(* Logix 5000 project; controller Project1Template vendor 1 type 14 code 151 rev 33.12; software revision 33.01 *)

TASK MainTask (continuous, watchdog 500 ms) : MainProgram

MODULES
   Local : vendor 1 type 14 code 151 (Compact 0, rev 33.12)
      Discrete_IO : Embedded (Compact 1, rev 3.1, Output RPI 20 ms)
      Analog_IO : Embedded (Compact 2, rev 1.1, Output RPI 80 ms)
      Counters : Embedded (Compact 3, rev 1.1, Output RPI 20 ms)
END_MODULES

TYPE SHIFT_DATA :
STRUCT
   COMPLETED : DINT;
   PASSED : DINT;
   FAILED : DINT;
   EFFICIENT : REAL;
END_STRUCT
END_TYPE

ADD_ON_INSTRUCTION AOI_SIM_2PosCyl_ExtRet   (* revision 1.0 *)
VAR_OUTPUT
   Animation : DINT; {visible}
END_VAR
VAR_INPUT
   TravelTime : DINT; {required}
   Extend_Output : BOOL; {required}
   Retract_Output : BOOL; {required}
END_VAR
VAR_OUTPUT
   Extend_Sensor : BOOL; {access Read Only, required}
   Retract_Sensor : BOOL; {access Read Only, required}
END_VAR
VAR_INPUT
   MCR : BOOL; {required}
   SingleSolenoidExtend : BOOL; {required}
   SingleSolenoidRetract : BOOL; {required}
   Retract_ValvePB : BOOL;
   Extend_ValvePB : BOOL;
END_VAR
VAR
   Extend_ScanCount : DINT;
   Retract_ScanCount : DINT; {access None}
   Extend_Timer : TIMER := (PRE := 500); {access None}
   Retract_Timer : TIMER := (PRE := 500); {access None}
   Retracted : BOOL; {access None}
   Extended : BOOL; {access None}
   Retract : BOOL; {access None}
   Extend : BOOL; {access None}
END_VAR

ROUTINE Logic   (* ladder *)
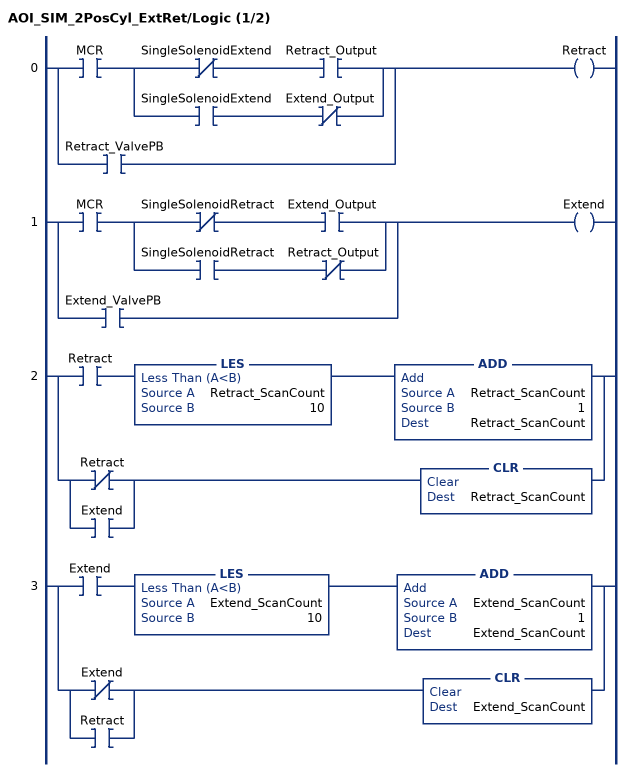
   0: [XIC(MCR) [XIO(SingleSolenoidExtend) XIC(Retract_Output) ,XIC(SingleSolenoidExtend) XIO(Extend_Output) ] ,XIC(Retract_ValvePB) ]OTE(Retract);
   1: [XIC(MCR) [XIO(SingleSolenoidRetract) XIC(Extend_Output) ,XIC(SingleSolenoidRetract) XIO(Retract_Output) ] ,XIC(Extend_ValvePB) ]OTE(Extend);
   2: [XIC(Retract) LES(Retract_ScanCount,10) ADD(Retract_ScanCount,1,Retract_ScanCount) ,[XIO(Retract) ,XIC(Extend) ] CLR(Retract_ScanCount) ];
   3: [XIC(Extend) LES(Extend_ScanCount,10) ADD(Extend_ScanCount,1,Extend_ScanCount) ,[XIO(Extend) ,XIC(Retract) ] CLR(Extend_ScanCount) ];
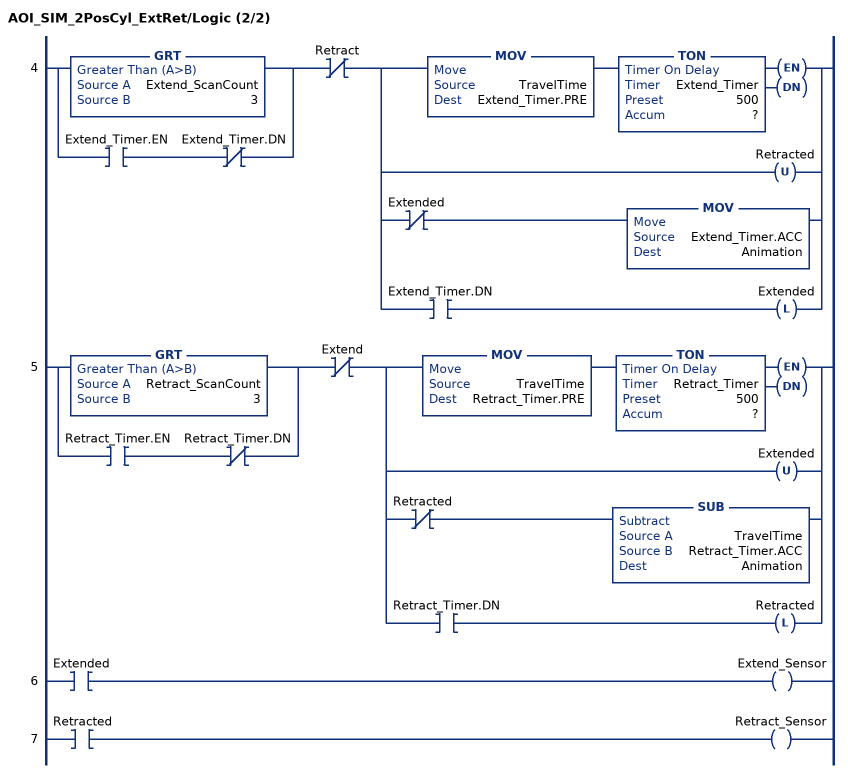
   4: [GRT(Extend_ScanCount,3) ,XIC(Extend_Timer.EN) XIO(Extend_Timer.DN) ]XIO(Retract)[MOV(TravelTime,Extend_Timer.PRE) TON(Extend_Timer,?,?) ,OTU(Retracted) ,XIO(Extended) MOV(Extend_Timer.ACC,Animation) ,XIC(Extend_Timer.DN) OTL(Extended) ];
   5: [GRT(Retract_ScanCount,3) ,XIC(Retract_Timer.EN) XIO(Retract_Timer.DN) ]XIO(Extend)[MOV(TravelTime,Retract_Timer.PRE) TON(Retract_Timer,?,?) ,OTU(Extended) ,XIO(Retracted) SUB(TravelTime,Retract_Timer.ACC,Animation) ,XIC(Retract_Timer.DN) OTL(Retracted) ];
   6: XIC(Extended)OTE(Extend_Sensor);
   7: XIC(Retracted)OTE(Retract_Sensor);
END_ROUTINE
END_ADD_ON_INSTRUCTION

ADD_ON_INSTRUCTION AOI_SIM_RandomDelay   (* revision 1.0 *)
VAR_INPUT
   Activate : BOOL; {access None}
   Target : DINT; {access None, required}
   Tolerance : DINT; {access None, required}
   PulseOutputTime : DINT; {access None, required}
END_VAR
VAR_OUTPUT
   DN : BOOL; {access Read Only, required}
END_VAR
VAR_INPUT
   DeActivate : BOOL; {access None}
END_VAR
VAR_OUTPUT
   TimingFirstHalf : BOOL; {access Read Only}
   TimingLastHalf : BOOL; {access Read Only}
   AccumlatedTime : DINT; {access Read Only}
   TT : BOOL; {access Read Only}
END_VAR
VAR
   StartTimerPulse : BOOL; {access None}
   StartTimerONS : BOOL; {access None}
   RandomIntermediate : DINT; {access None}
   RandomNumber : DINT; {access None}
   RandomPresetTime : DINT; {access None}
   RandomTimer : TIMER; {access None}
   PulseOutput : TIMER; {access None}
   Time50Percent : DINT; {access None}
END_VAR

ROUTINE Logic   (* ladder *)
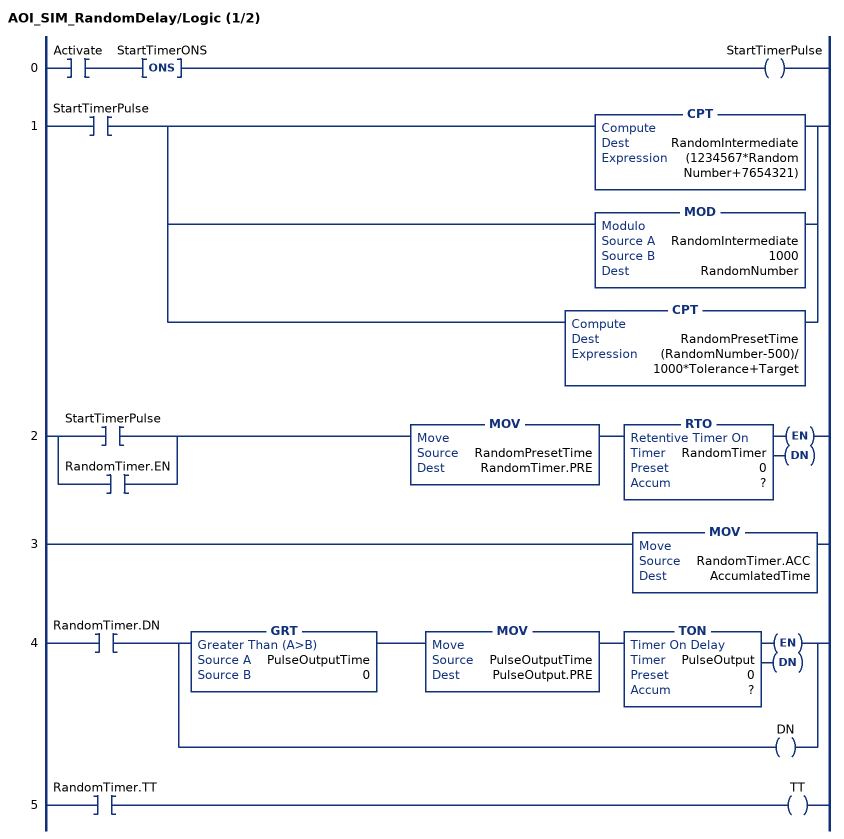
   0: XIC(Activate)ONS(StartTimerONS)OTE(StartTimerPulse);
   1: XIC(StartTimerPulse)[CPT(RandomIntermediate,(1234567*RandomNumber+7654321)) ,MOD(RandomIntermediate,1000,RandomNumber) ,CPT(RandomPresetTime,(RandomNumber-500)/1000*Tolerance+Target) ];
   2: [XIC(StartTimerPulse) ,XIC(RandomTimer.EN) ]MOV(RandomPresetTime,RandomTimer.PRE)RTO(RandomTimer,?,?);
   3: MOV(RandomTimer.ACC,AccumlatedTime);
   4: XIC(RandomTimer.DN)[GRT(PulseOutputTime,0) MOV(PulseOutputTime,PulseOutput.PRE) TON(PulseOutput,?,?) ,OTE(DN) ];
   5: XIC(RandomTimer.TT)OTE(TT);
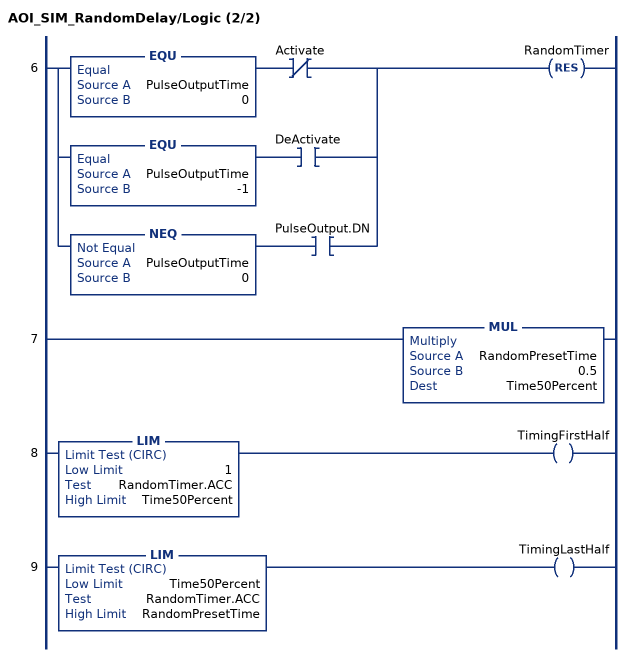
   6: [EQU(PulseOutputTime,0) XIO(Activate) ,EQU(PulseOutputTime,-1) XIC(DeActivate) ,NEQ(PulseOutputTime,0) XIC(PulseOutput.DN) ]RES(RandomTimer);
   7: MUL(RandomPresetTime,0.5,Time50Percent);
   8: LIM(1,RandomTimer.ACC,Time50Percent)OTE(TimingFirstHalf);
   9: LIM(Time50Percent,RandomTimer.ACC,RandomPresetTime)OTE(TimingLastHalf);
END_ROUTINE
END_ADD_ON_INSTRUCTION

ADD_ON_INSTRUCTION AOI_SIMAnalogSensor   (* revision 1.0 *)
VAR_IN_OUT
   Sensor : REAL; {required}
END_VAR
VAR_INPUT
   RampUpTime : DINT; {required}
   RampDwnTime : DINT; {required}
   Min : REAL; {required}
   Max : REAL; {required}
   Target : REAL; {required}
   Tolerance : REAL; {required}
   Fluctuation : REAL; {access None, required}
   Activate : BOOL; {access None}
END_VAR
VAR
   RampUpTimer : TIMER; {access None}
   RampDwnTimer : TIMER; {access None}
   FluctuateTimer : TIMER; {access None}
   FluctuateONS : BOOL; {access None}
   CurrentValue : REAL; {access Read Only}
   RampDwnTriggerONS : BOOL; {access Read Only}
   RampDwnTriggerPulse : BOOL; {access Read Only}
   RampUpTriggerONS : BOOL; {access Read Only}
   RampUpTriggerPulse : BOOL; {access Read Only}
   RandomNumber : DINT; {access Read Only}
   RandomTarget : REAL; {access Read Only}
   RandomIntermediate : DINT; {access Read Only}
   ScaledRampDwnTime : REAL; {access Read Only}
   ScaledRampUpTime : REAL; {access Read Only}
   Fluctuate : BOOL; {access None}
END_VAR

ROUTINE Logic   (* ladder *)
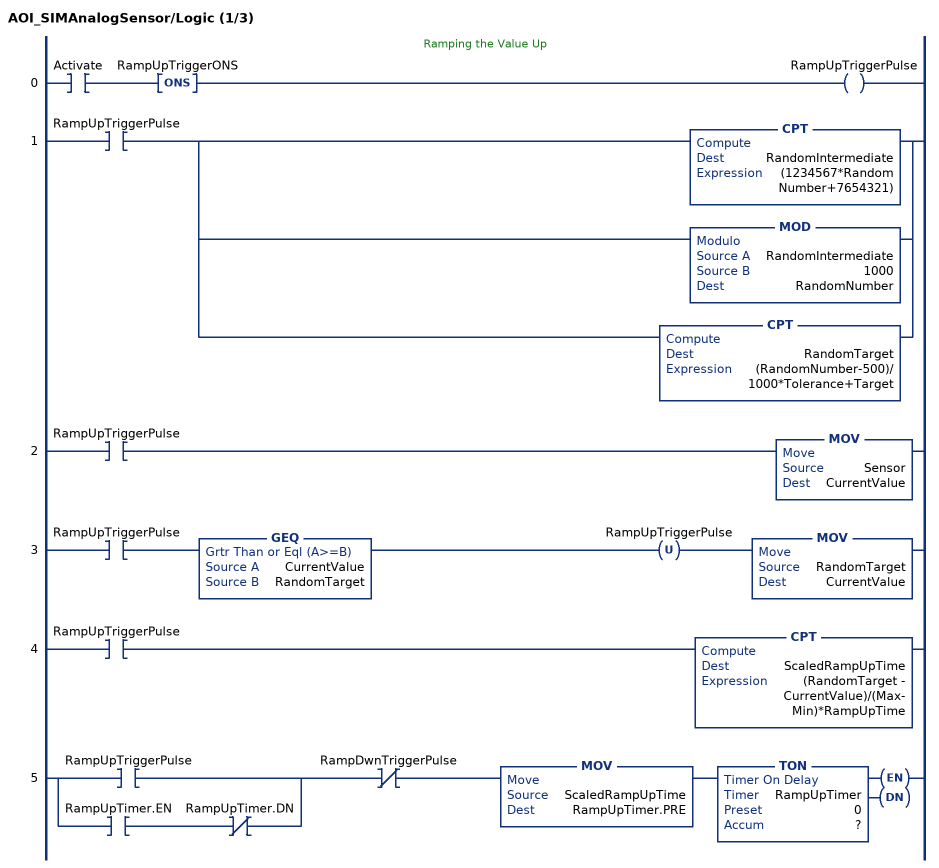
   // Ramping the Value Up
   0: XIC(Activate)ONS(RampUpTriggerONS)OTE(RampUpTriggerPulse);
   1: XIC(RampUpTriggerPulse)[CPT(RandomIntermediate,(1234567*RandomNumber+7654321)) ,MOD(RandomIntermediate,1000,RandomNumber) ,CPT(RandomTarget,(RandomNumber-500)/1000*Tolerance+Target) ];
   2: XIC(RampUpTriggerPulse)MOV(Sensor,CurrentValue);
   3: XIC(RampUpTriggerPulse)GEQ(CurrentValue,RandomTarget)OTU(RampUpTriggerPulse)MOV(RandomTarget,CurrentValue);
   4: XIC(RampUpTriggerPulse)CPT(ScaledRampUpTime,(RandomTarget - CurrentValue)/(Max-Min)*RampUpTime);
   5: [XIC(RampUpTriggerPulse) ,XIC(RampUpTimer.EN) XIO(RampUpTimer.DN) ]XIO(RampDwnTriggerPulse)MOV(ScaledRampUpTime,RampUpTimer.PRE)TON(RampUpTimer,?,?);
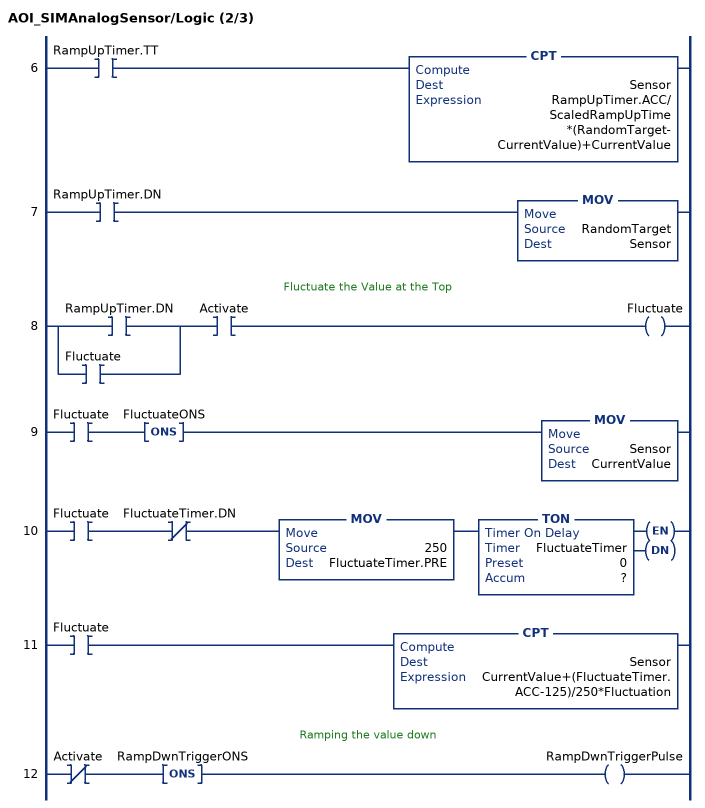
   6: XIC(RampUpTimer.TT)CPT(Sensor,RampUpTimer.ACC/ScaledRampUpTime *(RandomTarget-CurrentValue)+CurrentValue);
   7: XIC(RampUpTimer.DN)MOV(RandomTarget,Sensor);
   // Fluctuate the Value at the Top
   8: [XIC(RampUpTimer.DN) ,XIC(Fluctuate) ]XIC(Activate)OTE(Fluctuate);
   9: XIC(Fluctuate)ONS(FluctuateONS)MOV(Sensor,CurrentValue);
   10: XIC(Fluctuate)XIO(FluctuateTimer.DN)MOV(250,FluctuateTimer.PRE)TON(FluctuateTimer,?,?);
   11: XIC(Fluctuate)CPT(Sensor,CurrentValue+(FluctuateTimer.ACC-125)/250*Fluctuation);
   // Ramping the value down
   12: XIO(Activate)ONS(RampDwnTriggerONS)OTE(RampDwnTriggerPulse);
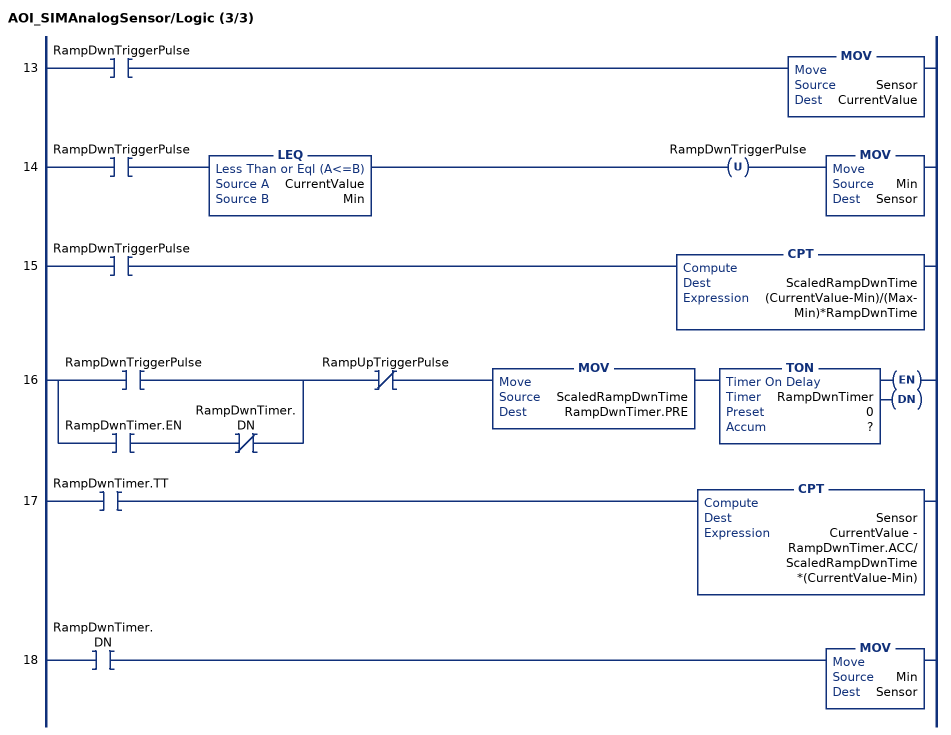
   13: XIC(RampDwnTriggerPulse)MOV(Sensor,CurrentValue);
   14: XIC(RampDwnTriggerPulse)LEQ(CurrentValue,Min)OTU(RampDwnTriggerPulse)MOV(Min,Sensor);
   15: XIC(RampDwnTriggerPulse)CPT(ScaledRampDwnTime,(CurrentValue-Min)/(Max-Min)*RampDwnTime);
   16: [XIC(RampDwnTriggerPulse) ,XIC(RampDwnTimer.EN) XIO(RampDwnTimer.DN) ]XIO(RampUpTriggerPulse)MOV(ScaledRampDwnTime,RampDwnTimer.PRE)TON(RampDwnTimer,?,?);
   17: XIC(RampDwnTimer.TT)CPT(Sensor,CurrentValue - RampDwnTimer.ACC/ScaledRampDwnTime *(CurrentValue-Min));
   18: XIC(RampDwnTimer.DN)MOV(Min,Sensor);
END_ROUTINE
END_ADD_ON_INSTRUCTION

VAR_GLOBAL   (* controller tags *)
   A_EXT_TMR : TIMER := (PRE := 10000);
   A_RET_TMR : TIMER := (PRE := 10000);
   ADD12 : DINT;
   ADD123 : DINT;
   ADD123FAIL : DINT;
   ADD123PASS : DINT;
   ADD12FAIL : DINT;
   ADD12PASS : DINT;
   ALLFAILONES : BOOL;
   AVERAGE1 : CONTROL := (LEN := 50);
   AVERAGECNTRL : CONTROL := (LEN := 50);
   B_EXT_TMR : TIMER := (PRE := 10000);
   B_RET_TMR : TIMER := (PRE := 10000);
   C_EXT_TMR : TIMER := (PRE := 10000);
   C_RET_TMR : TIMER := (PRE := 10000);
   CHANGED : BOOL;
   CHANGEONS : BOOL;
   CURRENT_SHIFT : SHIFT_DATA;
   DATASHIFT : BOOL;
   EFFICIENCY : REAL;
   END_SHIFT_PB : BOOL;
   EStop : BOOL;
   EXTRA_TIME : TIMER := (PRE := 120000);
   F1_AVERAGE : REAL;
   F1_Count : COUNTER;
   F1_FAIL : COUNTER;
   F1_PASS : COUNTER;
   F1_TEMP_TORQUE : DINT[50];
   F1_TORQUE : REAL[50];
   F2_Count : COUNTER;
   F2_FAIL : COUNTER;
   F2_PASS : COUNTER;
   F3_Count : COUNTER;
   F3_FAIL : COUNTER;
   F3_PASS : COUNTER;
   F4_Count : COUNTER;
   F4_FAIL : COUNTER;
   F4_PASS : COUNTER;
   F_ALL_CTR : COUNTER := (ACC := 1);
   FAILONS1 : BOOL;
   FAILONS2 : BOOL;
   FAILONS3 : BOOL;
   FAILONS4 : BOOL;
   FASTEN_AllComplete : BOOL;
   FASTEN_AllTorquesFail : BOOL;
   FASTEN_AllTorquesPass : BOOL;
   FASTEN_F1Complete : BOOL;
   FASTEN_F1Complete_ONS : BOOL;
   FASTEN_F1Torque : REAL;
   FASTEN_F1TorqueFail : BOOL;
   FASTEN_F1TorquePass : BOOL;
   FASTEN_F2Complete : BOOL;
   FASTEN_F2Complete_ONS : BOOL;
   FASTEN_F2Torque : REAL;
   FASTEN_F2TorqueFail : BOOL;
   FASTEN_F2TorquePass : BOOL;
   FASTEN_F3Complete : BOOL;
   FASTEN_F3Complete_ONS : BOOL;
   FASTEN_F3Torque : REAL;
   FASTEN_F3TorqueFail : BOOL;
   FASTEN_F3TorquePass : BOOL;
   FASTEN_F4Complete : BOOL;
   FASTEN_F4Complete_ONS : BOOL;
   FASTEN_F4Torque : REAL;
   FASTEN_F4TorqueFail : BOOL;
   FASTEN_F4TorquePass : BOOL;
   FASTEN_TorqueFeedback : REAL := 20.050001;
   FAULTRESET_PB : BOOL;
   FAULTS : DINT;
   FAULTSIND : BOOL;
   FIX_EXT_TMR : TIMER := (PRE := 10000);
   FIX_RET_TMR : TIMER := (PRE := 10000);
   FIXTURE_AllPartsPresent : BOOL := 1;
   FIXTURE_AtHomePos : BOOL := 1;
   FIXTURE_Empty : BOOL;
   FIXTURE_PartsSecured : BOOL;
   FIXTURE_PartsSecuredTmr : TIMER := (PRE := 500);
   FromHMI_ExtClampA_PB : BOOL;
   FromHMI_ExtClampB_PB : BOOL;
   FromHMI_ExtClampC_PB : BOOL;
   FromHMI_ExtFixture_PB : BOOL;
   FromHMI_F1LowLim : REAL := 75.0;
   FromHMI_F1UppLim : REAL := 95.0;
   FromHMI_F2LowLim : REAL := 75.0;
   FromHMI_F2UppLim : REAL := 85.0;
   FromHMI_F3LowLim : REAL := 75.0;
   FromHMI_F3UppLim : REAL := 85.0;
   FromHMI_F4LowLim : REAL := 75.0;
   FromHMI_F4UppLim : REAL := 95.0;
   FromHMI_RetClampA_PB : BOOL;
   FromHMI_RetClampB_PB : BOOL;
   FromHMI_RetClampC_PB : BOOL;
   FromHMI_RetFixture_PB : BOOL;
   FROMHMI_SCREEN : DINT;
   FromHMI_StartPB : BOOL;
   FromHMI_StopPB : BOOL := 1;
   FromRbt_ClearOfFixture : BOOL := 1;
   FromRbt_Fasten1Complete : BOOL;
   FromRbt_Fasten2Complete : BOOL;
   FromRbt_Fasten3Complete : BOOL;
   FromRbt_Fasten4Complete : BOOL;
   HomePB : BOOL;
   I1 : INT := 20318;
        .10   // Part Present C Sensor
        .11   // Part Present D Sensor
        .14   // Light Curtain Safety Circuit
        .0   // Fixture at Robot Limit Switch
        .1   // Fixture at Operator Limit Switch
        .2   // Clamp A Retracted Limit Switch
        .3   // Clamp B Retracted Limit Switch
        .4   // Clamp C Retracted Limit Switch
        .8   // Part Present A Sensor
        .9   // Part Present B Sensor
   I2_CHA : REAL := 4.01;   // Torque Sensor Input
   O3 : INT;
        .1   // Fixture Retract to Operator
        .3   // Clamp B Extend Solenoid
        .0   // Fixture Extend to Robot
        .2   // Clamp A Extend Solenoid
        .4   // Clamp C Extend Solenoid
   ONEHR : BOOL;
   ONS1 : BOOL;
   ONS2 : BOOL;
   ONS3 : BOOL;
   ONS4 : BOOL;
   RESET_STATS : BOOL;
   S1ON : BOOL;
   SCREENREQTMR : TIMER := (PRE := 1000);
   SHIFT1ONS : BOOL;
   SHIFT_CHANGE : BOOL;
   SHIFT_TIMER : TIMER := (PRE := 120000);
   SHIFTHISTORY : SHIFT_DATA[5];
   SHIFTONS : BOOL;
   STARTONS : BOOL;
   SYS_AutoModeActive : BOOL := 1;
   SYS_CycleActive : BOOL;
   SYS_ManualModeActive : BOOL;
   SYS_StartPBPulseTmr : TIMER := (PRE := 200);
   T1AVG : DINT;
   THREEHR : BOOL;
   TIME : REAL;
   TOHMI_CHANGEVALVE : BOOL;
   TOHMI_CHANGEWARNING : BOOL;
   TOHMI_SCREENREQ : DINT;
   ToRbt_Fasten1Start : BOOL;
   ToRbt_Fasten2Start : BOOL;
   ToRbt_Fasten3Start : BOOL;
   ToRbt_Fasten4Start : BOOL;
   TOTAL_PARTS_COMPLETE : DINT;
   TOTAL_PARTS_FAIL : DINT;
   TOTAL_PARTS_PASS : DINT;
   TWOHR : BOOL;
   VALVECTR : COUNTER;
   VALVEONS : BOOL;
   VALVEWARNING : DINT;
END_VAR

PROGRAM MainProgram   (* main routine MainRoutine *)
VAR
   SIM_ClampA : AOI_SIM_2PosCyl_ExtRet := (TravelTime := 1000, Retract_Sensor := 1, MCR := 1, SingleSolenoidExtend := 1);
   SIM_ClampB : AOI_SIM_2PosCyl_ExtRet := (TravelTime := 1250, Retract_Sensor := 1, MCR := 1, SingleSolenoidExtend := 1);
   SIM_ClampC : AOI_SIM_2PosCyl_ExtRet := (TravelTime := 1250, Retract_Sensor := 1, MCR := 1, SingleSolenoidExtend := 1);
   SIM_EmptyFixture : TIMER := (PRE := 15000);
   SIM_Fasten1 : AOI_SIM_RandomDelay := (Target := 2500, Tolerance := 750);
   SIM_Fasten2 : AOI_SIM_RandomDelay := (Target := 3500, Tolerance := 450);
   SIM_Fasten3 : AOI_SIM_RandomDelay := (Target := 4500, Tolerance := 250);
   SIM_Fasten4 : AOI_SIM_RandomDelay := (Target := 3750, Tolerance := 500);
   SIM_Fixture : AOI_SIM_2PosCyl_ExtRet := (TravelTime := 2000, Retract_Sensor := 1, MCR := 1);
   SIM_LightCurtainPartPlace : AOI_SIM_RandomDelay := (Target := 6000, Tolerance := 1500, PulseOutputTime := 50);
   SIM_LightCurtainPartRem : AOI_SIM_RandomDelay := (Target := 5000, Tolerance := 1000, PulseOutputTime := 50);
   SIM_NOP : BOOL;
   SIM_Oneshots : DINT := 1;
   SIM_OperatorWorking : AOI_SIM_RandomDelay := (Target := 4000, Tolerance := 2000, PulseOutputTime := 50);
   SIM_PP_OFF : AOI_SIM_RandomDelay := (Target := 2500, Tolerance := 1000, PulseOutputTime := 50);
   SIM_PPA_ON : AOI_SIM_RandomDelay := (Target := 1500, Tolerance := 500, PulseOutputTime := 50);
   SIM_PPB_ON : AOI_SIM_RandomDelay := (Target := 2000, Tolerance := 1000, PulseOutputTime := 50);
   SIM_PPC_ON : AOI_SIM_RandomDelay := (Target := 2500, Tolerance := 1000, PulseOutputTime := 50);
   SIM_PPD_ON : AOI_SIM_RandomDelay := (Target := 3000, Tolerance := 500, PulseOutputTime := 50);
   SIM_RobotClear : AOI_SIM_RandomDelay := (Target := 1200, Tolerance := 250, PulseOutputTime := 50);
   SIM_Torque : AOI_SIMAnalogSensor := (RampUpTime := 500, RampDwnTime := 50, Min := 4.01, Max := 19.99, Target := 15.0, Tolerance := 2.0, Fluctuation := 0.04);
END_VAR

ROUTINE EXTRAS   (* ladder *)
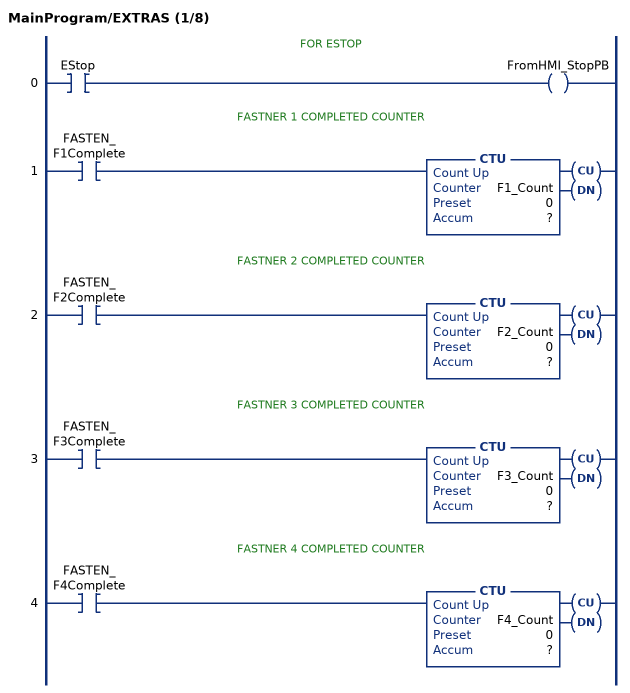
   // FOR ESTOP
   0: XIC(EStop)OTE(FromHMI_StopPB);
   // FASTNER 1 COMPLETED COUNTER
   1: XIC(FASTEN_F1Complete)CTU(F1_Count,?,?);
   // FASTNER 2 COMPLETED COUNTER
   2: XIC(FASTEN_F2Complete)CTU(F2_Count,?,?);
   // FASTNER 3 COMPLETED COUNTER
   3: XIC(FASTEN_F3Complete)CTU(F3_Count,?,?);
   // FASTNER 4 COMPLETED COUNTER
   4: XIC(FASTEN_F4Complete)CTU(F4_Count,?,?);
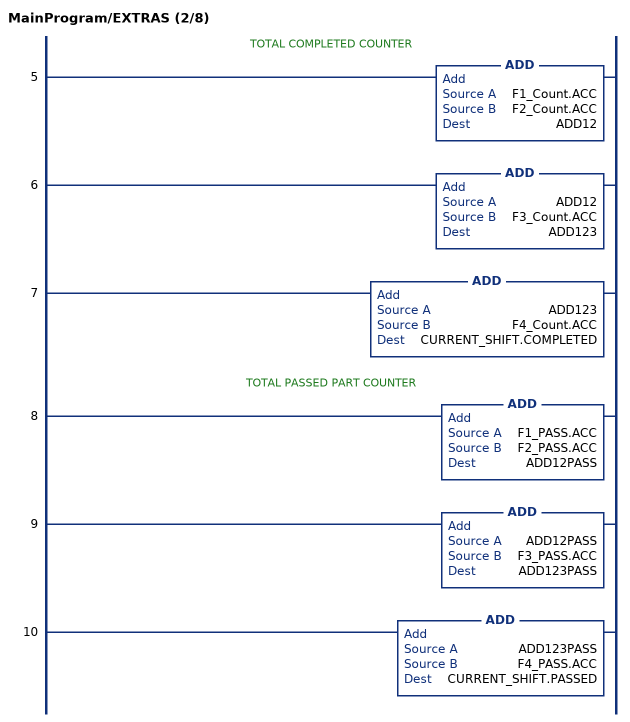
   // TOTAL COMPLETED COUNTER
   5: ADD(F1_Count.ACC,F2_Count.ACC,ADD12);
   6: ADD(ADD12,F3_Count.ACC,ADD123);
   7: ADD(ADD123,F4_Count.ACC,CURRENT_SHIFT.COMPLETED);
   // TOTAL PASSED PART COUNTER
   8: ADD(F1_PASS.ACC,F2_PASS.ACC,ADD12PASS);
   9: ADD(ADD12PASS,F3_PASS.ACC,ADD123PASS);
   10: ADD(ADD123PASS,F4_PASS.ACC,CURRENT_SHIFT.PASSED);
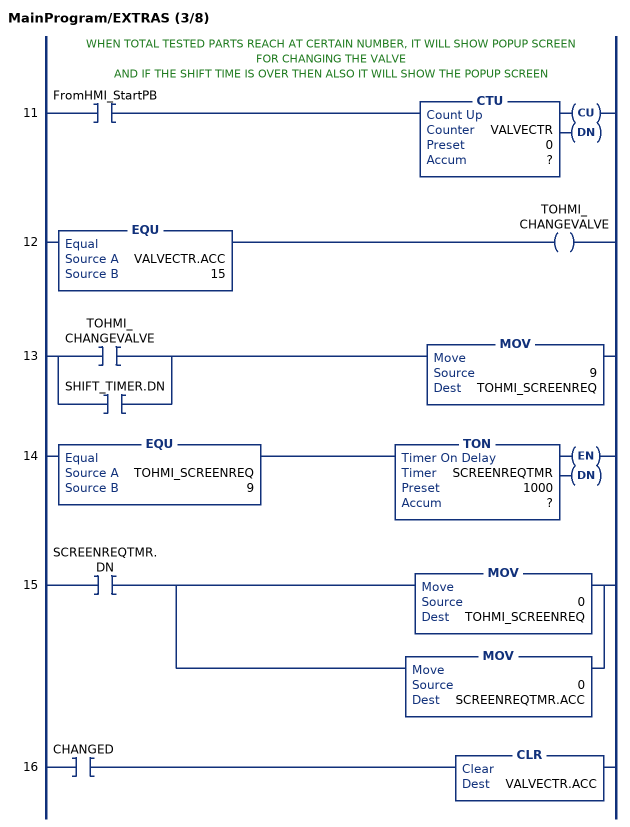
   // WHEN TOTAL TESTED PARTS REACH AT CERTAIN NUMBER, IT WILL SHOW POPUP SCREEN FOR CHANGING THE VALVE
   // AND IF THE SHIFT TIME IS OVER THEN ALSO IT WILL SHOW THE POPUP SCREEN
   11: XIC(FromHMI_StartPB)CTU(VALVECTR,?,?);
   12: EQU(VALVECTR.ACC,15)OTE(TOHMI_CHANGEVALVE);
   13: [XIC(TOHMI_CHANGEVALVE) ,XIC(SHIFT_TIMER.DN) ]MOV(9,TOHMI_SCREENREQ);
   14: EQU(TOHMI_SCREENREQ,9)TON(SCREENREQTMR,?,?);
   15: XIC(SCREENREQTMR.DN)[MOV(0,TOHMI_SCREENREQ) ,MOV(0,SCREENREQTMR.ACC) ];
   16: XIC(CHANGED)CLR(VALVECTR.ACC);
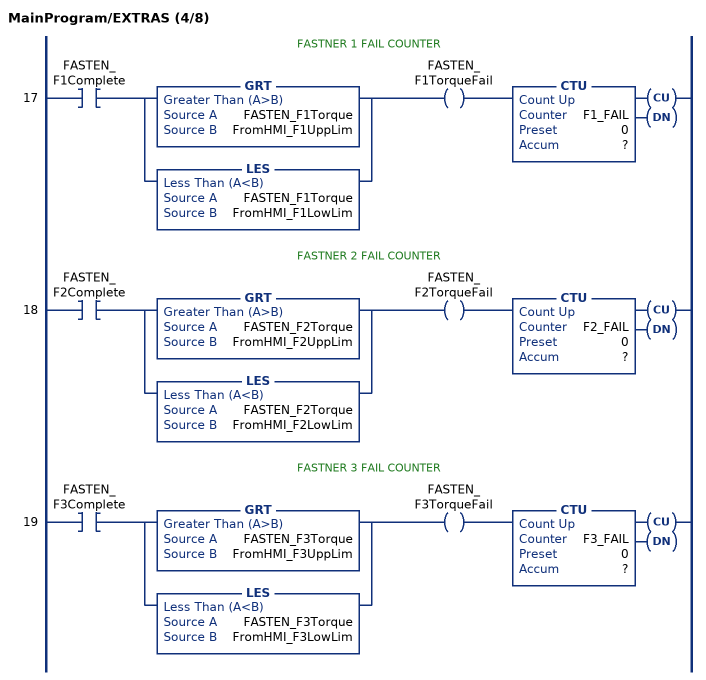
   // FASTNER 1 FAIL COUNTER
   17: XIC(FASTEN_F1Complete)[GRT(FASTEN_F1Torque,FromHMI_F1UppLim) ,LES(FASTEN_F1Torque,FromHMI_F1LowLim) ]OTE(FASTEN_F1TorqueFail)CTU(F1_FAIL,?,?);
   // FASTNER 2 FAIL COUNTER
   18: XIC(FASTEN_F2Complete)[GRT(FASTEN_F2Torque,FromHMI_F2UppLim) ,LES(FASTEN_F2Torque,FromHMI_F2LowLim) ]OTE(FASTEN_F2TorqueFail)CTU(F2_FAIL,?,?);
   // FASTNER 3 FAIL COUNTER
   19: XIC(FASTEN_F3Complete)[GRT(FASTEN_F3Torque,FromHMI_F3UppLim) ,LES(FASTEN_F3Torque,FromHMI_F3LowLim) ]OTE(FASTEN_F3TorqueFail)CTU(F3_FAIL,?,?);
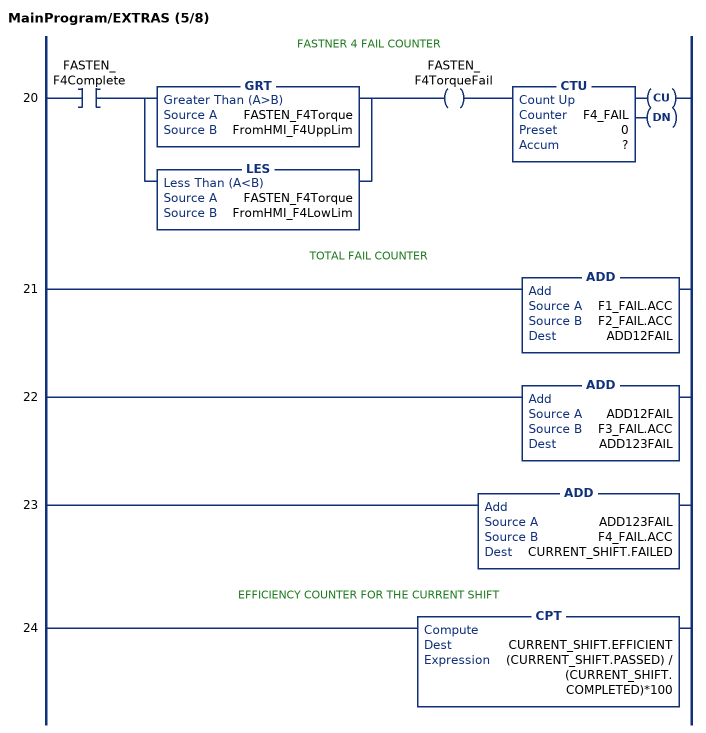
   // FASTNER 4 FAIL COUNTER
   20: XIC(FASTEN_F4Complete)[GRT(FASTEN_F4Torque,FromHMI_F4UppLim) ,LES(FASTEN_F4Torque,FromHMI_F4LowLim) ]OTE(FASTEN_F4TorqueFail)CTU(F4_FAIL,?,?);
   // TOTAL FAIL COUNTER
   21: ADD(F1_FAIL.ACC,F2_FAIL.ACC,ADD12FAIL);
   22: ADD(ADD12FAIL,F3_FAIL.ACC,ADD123FAIL);
   23: ADD(ADD123FAIL,F4_FAIL.ACC,CURRENT_SHIFT.FAILED);
   // EFFICIENCY COUNTER FOR THE CURRENT SHIFT
   24: CPT(CURRENT_SHIFT.EFFICIENT,(CURRENT_SHIFT.PASSED) / (CURRENT_SHIFT.COMPLETED)*100);
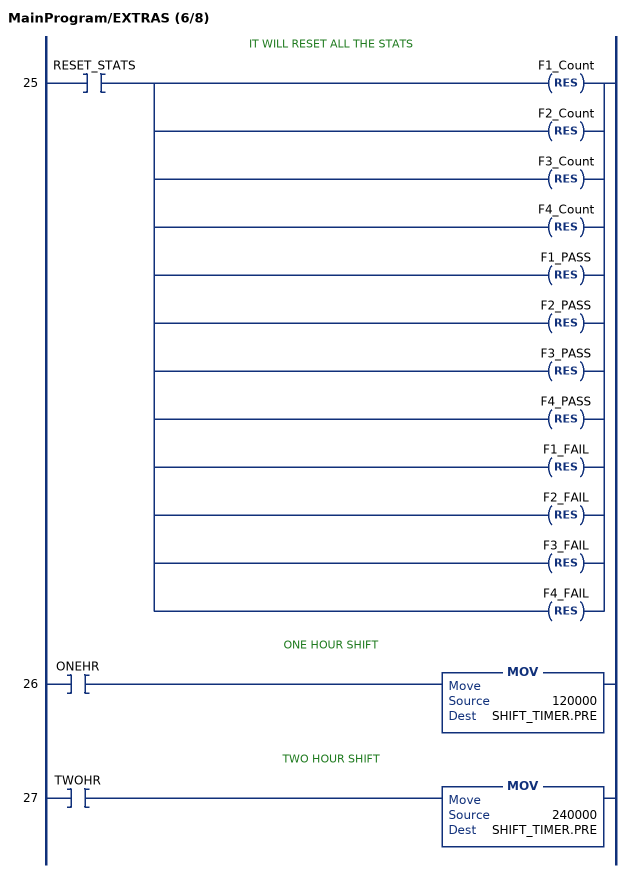
   // IT WILL RESET ALL THE STATS
   25: XIC(RESET_STATS)[RES(F1_Count) ,RES(F2_Count) ,RES(F3_Count) ,RES(F4_Count) ,RES(F1_PASS) ,RES(F2_PASS) ,RES(F3_PASS) ,RES(F4_PASS) ,RES(F1_FAIL) ,RES(F2_FAIL) ,RES(F3_FAIL) ,RES(F4_FAIL) ];
   // ONE HOUR SHIFT
   26: XIC(ONEHR)MOV(120000,SHIFT_TIMER.PRE);
   // TWO HOUR SHIFT
   27: XIC(TWOHR)MOV(240000,SHIFT_TIMER.PRE);
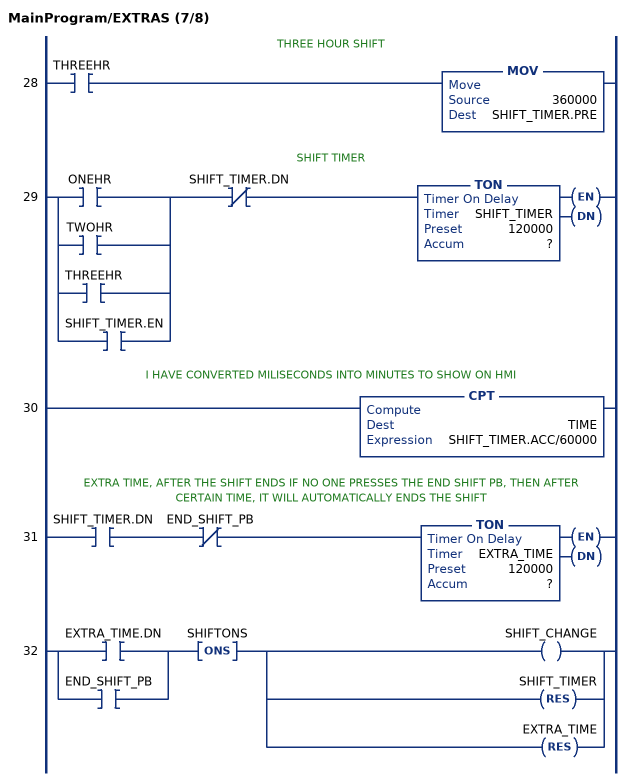
   // THREE HOUR SHIFT
   28: XIC(THREEHR)MOV(360000,SHIFT_TIMER.PRE);
   // SHIFT TIMER
   29: [[XIC(ONEHR) ,XIC(TWOHR) ,XIC(THREEHR) ] ,XIC(SHIFT_TIMER.EN) ]XIO(SHIFT_TIMER.DN)TON(SHIFT_TIMER,?,?);
   // I HAVE CONVERTED MILISECONDS INTO MINUTES TO SHOW ON HMI
   30: CPT(TIME,SHIFT_TIMER.ACC/60000);
   // EXTRA TIME, AFTER THE SHIFT ENDS IF NO ONE PRESSES THE END SHIFT PB, THEN AFTER CERTAIN TIME, IT WILL AUTOMATICALLY ENDS THE SHIFT
   31: XIC(SHIFT_TIMER.DN)XIO(END_SHIFT_PB)TON(EXTRA_TIME,?,?);
   32: [XIC(EXTRA_TIME.DN) ,XIC(END_SHIFT_PB) ]ONS(SHIFTONS)[OTE(SHIFT_CHANGE) ,RES(SHIFT_TIMER) ,RES(EXTRA_TIME) ];
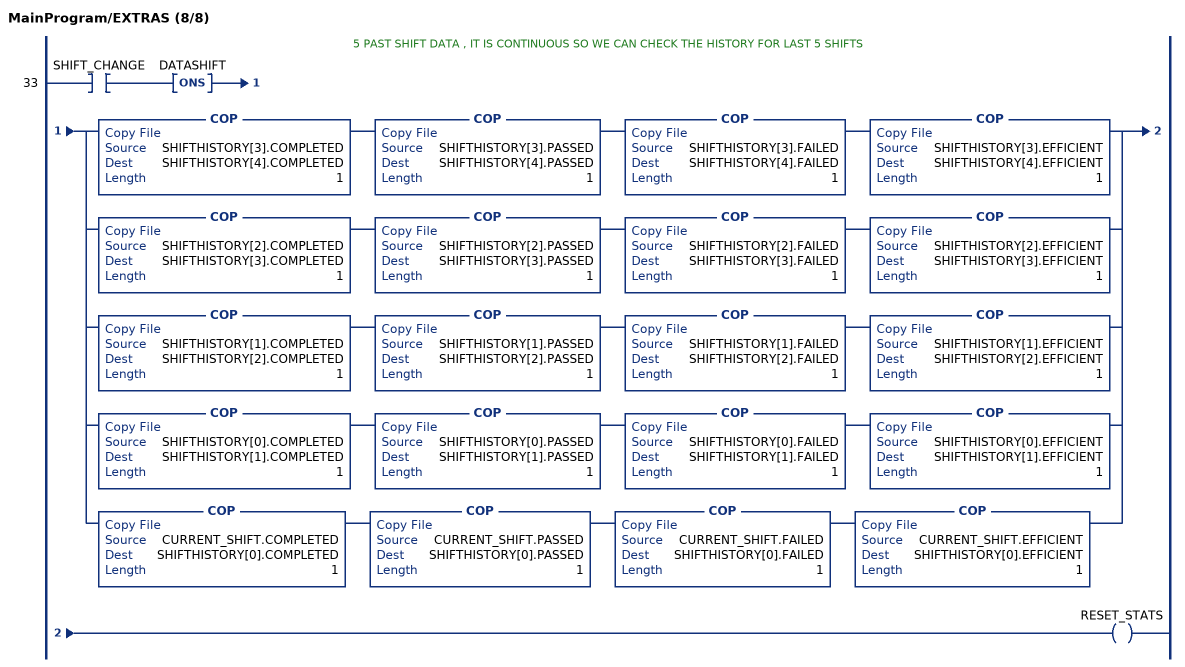
   // 5 PAST SHIFT DATA , IT IS CONTINUOUS SO WE CAN CHECK THE HISTORY FOR LAST 5 SHIFTS
   33: XIC(SHIFT_CHANGE)ONS(DATASHIFT)[COP(SHIFTHISTORY[3].COMPLETED,SHIFTHISTORY[4].COMPLETED,1) COP(SHIFTHISTORY[3].PASSED,SHIFTHISTORY[4].PASSED,1) COP(SHIFTHISTORY[3].FAILED,SHIFTHISTORY[4].FAILED,1) COP(SHIFTHISTORY[3].EFFICIENT,SHIFTHISTORY[4].EFFICIENT,1) ,COP(SHIFTHISTORY[2].COMPLETED,SHIFTHISTORY[3].COMPLETED,1) COP(SHIFTHISTORY[2].PASSED,SHIFTHISTORY[3].PASSED,1) COP(SHIFTHISTORY[2].FAILED,SHIFTHISTORY[3].FAILED,1) COP(SHIFTHISTORY[2].EFFICIENT,SHIFTHISTORY[3].EFFICIENT,1) ,COP(SHIFTHISTORY[1].COMPLETED,SHIFTHISTORY[2].COMPLETED,1) COP(SHIFTHISTORY[1].PASSED,SHIFTHISTORY[2].PASSED,1) COP(SHIFTHISTORY[1].FAILED,SHIFTHISTORY[2].FAILED,1) COP(SHIFTHISTORY[1].EFFICIENT,SHIFTHISTORY[2].EFFICIENT,1) ,COP(SHIFTHISTORY[0].COMPLETED,SHIFTHISTORY[1].COMPLETED,1) COP(SHIFTHISTORY[0].PASSED,SHIFTHISTORY[1].PASSED,1) COP(SHIFTHISTORY[0].FAILED,SHIFTHISTORY[1].FAILED,1) COP(SHIFTHISTORY[0].EFFICIENT,SHIFTHISTORY[1].EFFICIENT,1) ,COP(CURRENT_SHIFT.COMPLETED,SHIFTHISTORY[0].COMPLETED,1) COP(CURRENT_SHIFT.PASSED,SHIFTHISTORY[0].PASSED,1) COP(CURRENT_SHIFT.FAILED,SHIFTHISTORY[0].FAILED,1) COP(CURRENT_SHIFT.EFFICIENT,SHIFTHISTORY[0].EFFICIENT,1) ]OTE(RESET_STATS);
END_ROUTINE

ROUTINE FAULTS   (* ladder *)
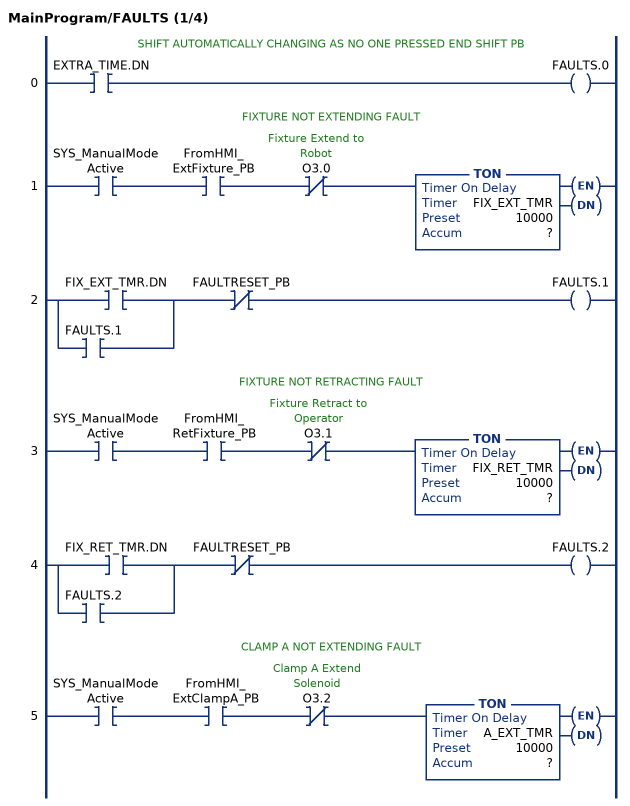
   // SHIFT AUTOMATICALLY CHANGING AS NO ONE PRESSED END SHIFT PB
   0: XIC(EXTRA_TIME.DN)OTE(FAULTS.0);
   // FIXTURE NOT EXTENDING FAULT
   1: XIC(SYS_ManualModeActive)XIC(FromHMI_ExtFixture_PB)XIO(O3.0)TON(FIX_EXT_TMR,?,?);
   2: [XIC(FIX_EXT_TMR.DN) ,XIC(FAULTS.1) ]XIO(FAULTRESET_PB)OTE(FAULTS.1);
   // FIXTURE NOT RETRACTING FAULT
   3: XIC(SYS_ManualModeActive)XIC(FromHMI_RetFixture_PB)XIO(O3.1)TON(FIX_RET_TMR,?,?);
   4: [XIC(FIX_RET_TMR.DN) ,XIC(FAULTS.2) ]XIO(FAULTRESET_PB)OTE(FAULTS.2);
   // CLAMP A NOT EXTENDING FAULT
   5: XIC(SYS_ManualModeActive)XIC(FromHMI_ExtClampA_PB)XIO(O3.2)TON(A_EXT_TMR,?,?);
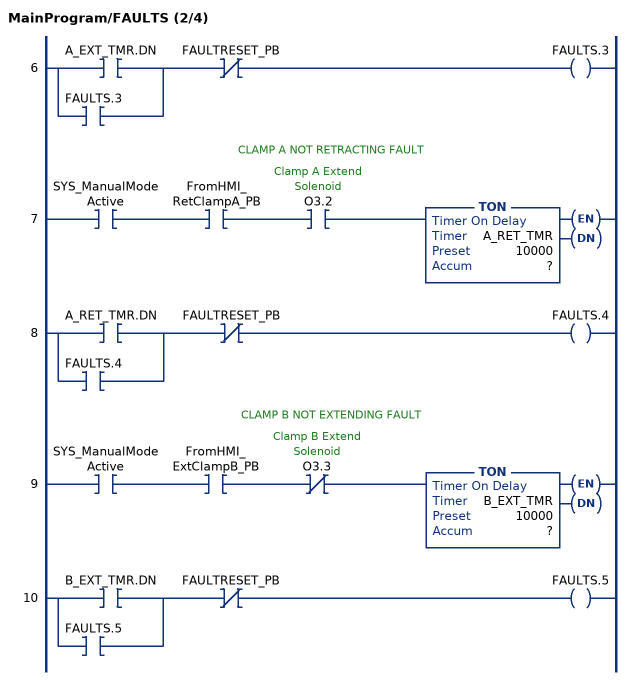
   6: [XIC(A_EXT_TMR.DN) ,XIC(FAULTS.3) ]XIO(FAULTRESET_PB)OTE(FAULTS.3);
   // CLAMP A NOT RETRACTING FAULT
   7: XIC(SYS_ManualModeActive)XIC(FromHMI_RetClampA_PB)XIC(O3.2)TON(A_RET_TMR,?,?);
   8: [XIC(A_RET_TMR.DN) ,XIC(FAULTS.4) ]XIO(FAULTRESET_PB)OTE(FAULTS.4);
   // CLAMP B NOT EXTENDING FAULT
   9: XIC(SYS_ManualModeActive)XIC(FromHMI_ExtClampB_PB)XIO(O3.3)TON(B_EXT_TMR,?,?);
   10: [XIC(B_EXT_TMR.DN) ,XIC(FAULTS.5) ]XIO(FAULTRESET_PB)OTE(FAULTS.5);
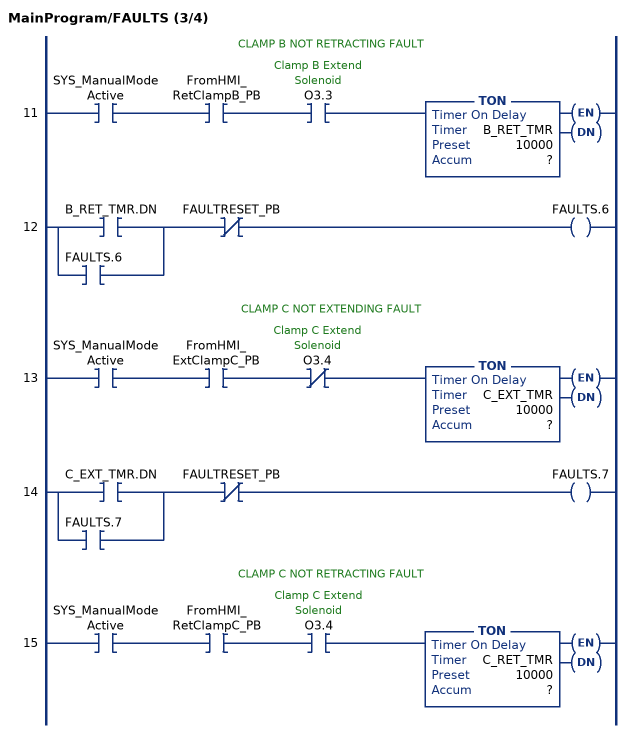
   // CLAMP B NOT RETRACTING FAULT
   11: XIC(SYS_ManualModeActive)XIC(FromHMI_RetClampB_PB)XIC(O3.3)TON(B_RET_TMR,?,?);
   12: [XIC(B_RET_TMR.DN) ,XIC(FAULTS.6) ]XIO(FAULTRESET_PB)OTE(FAULTS.6);
   // CLAMP C NOT EXTENDING FAULT
   13: XIC(SYS_ManualModeActive)XIC(FromHMI_ExtClampC_PB)XIO(O3.4)TON(C_EXT_TMR,?,?);
   14: [XIC(C_EXT_TMR.DN) ,XIC(FAULTS.7) ]XIO(FAULTRESET_PB)OTE(FAULTS.7);
   // CLAMP C NOT RETRACTING FAULT
   15: XIC(SYS_ManualModeActive)XIC(FromHMI_RetClampC_PB)XIC(O3.4)TON(C_RET_TMR,?,?);
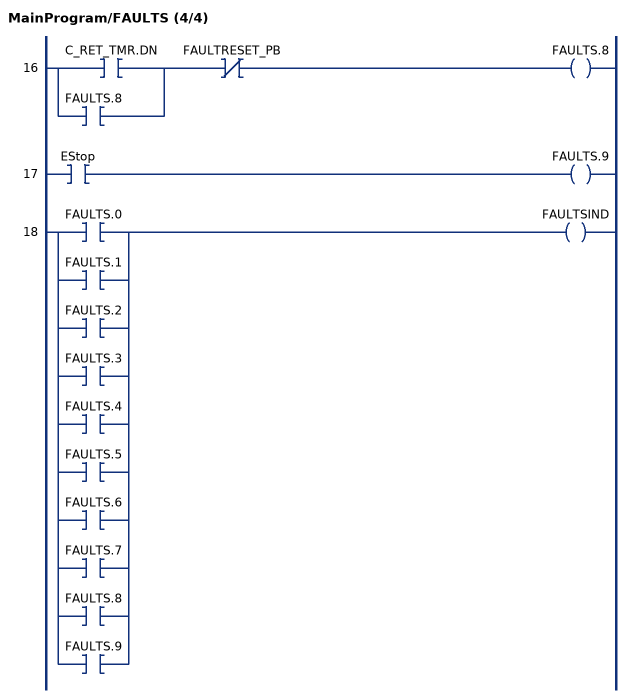
   16: [XIC(C_RET_TMR.DN) ,XIC(FAULTS.8) ]XIO(FAULTRESET_PB)OTE(FAULTS.8);
   17: XIC(EStop)OTE(FAULTS.9);
   18: [XIC(FAULTS.0) ,XIC(FAULTS.1) ,XIC(FAULTS.2) ,XIC(FAULTS.3) ,XIC(FAULTS.4) ,XIC(FAULTS.5) ,XIC(FAULTS.6) ,XIC(FAULTS.7) ,XIC(FAULTS.8) ,XIC(FAULTS.9) ]OTE(FAULTSIND);
END_ROUTINE
